{attribute 'GeneratedUsingTerminal: AT2050-0501-0022'}
{attribute addProperty BoxType "AT2050-0501-0022"}
{attribute addProperty Id "A_0082_AT2002_5250_0019_AT2002_5250AT2002_33A3DF1B80"}
{attribute addProperty CRC "3829779776"}
{attribute addProperty Size "80"}
TYPE A_0070_AT2050_0501_0022_AT2050_0501_E445CD40 EXTENDS AT2050_2EA6C9BF :
STRUCT
	{attribute addProperty Name "A_0082_AT2002_5250_0019_AT2002_5250"}
	A_0082_AT2002_5250_0019_AT2002_5250 : AT2002_33A3DF1B;
END_STRUCT
END_TYPE

(* stored: Version 1.2.0.0, ProductVersion 3.1.4024.9
   DUT A_0070_AT2050_0501_0022_AT2050_0501_E445CD40: Id {40ad377d-4d51-4834-b692-1c5aefcdafb2} *)
